// TwinCAT 3 PLC project PRG_B_BaseDecorator
// Title: B_BaseDecorate
// Company: RafalOS
// Author: Rafał Osajda
// ProjectVersion: 0.0.0.3
// ProgramVersion: 3.1.4024.0
// libraries:
//   B_Base, * (RafalOS)
//   Tc2_Standard, * (Beckhoff Automation GmbH)
//   Tc2_System, * (Beckhoff Automation GmbH)
//   Tc3_Module, * (Beckhoff Automation GmbH)
// project tree:
//   / PlcTask.TcTTO
//   POUs Compilation/ PRG_Compilation.TcPOU
//   POUs/A03_FB_BaseLoggerElementDecorator/ FB_BaseLoggerElementDecoratorParent.TcPOU (not stored), ITF_BaseLoggerElementDecoratorParent.TcIO (not stored)
//   POUs/A04_FB_BaseComponentDecorator/ FB_BaseComponentDecoratorParent.TcPOU (not stored), ITF_BaseComponentDecoratorParent.TcIO
//   POUs/A05_FB_BaseControlElementDecorator/ FB_BaseControlElementDecoratorParent.TcPOU (not stored), ITF_BaseControlElementDecoratorParent.TcIO (not stored)
//   POUs/A06_FB_BaseGroupElementDecorator/ FB_BaseGroupElementDecoratorParent.TcPOU (not stored), ITF_BaseGroupElementDecoratorParent.TcIO
//   POUs/A07_FB_BaseTopElementDecorator/ FB_BaseTopElementDecoratorParent.TcPOU (not stored), ITF_BaseTopElementDecoratorParent.TcIO (not stored)

CONFIGURATION PRG_B_BaseDecorator
    RESOURCE PLC ON TwinCAT3
        TASK PlcTask(INTERVAL := T#10ms, PRIORITY := 20);
        PROGRAM PRG_Compilation WITH PlcTask : PRG_Compilation;
    END_RESOURCE
END_CONFIGURATION

// ---- POUs/A04_FB_BaseComponentDecorator/ITF_BaseComponentDecoratorParent.TcIO
INTERFACE ITF_BaseComponentDecoratorParent EXTENDS ITF_BaseComponent

END_INTERFACE

// ---- POUs/A06_FB_BaseGroupElementDecorator/ITF_BaseGroupElementDecoratorParent.TcIO
INTERFACE ITF_BaseGroupElementDecoratorParent EXTENDS ITF_BaseGroupElement

END_INTERFACE

// ---- POUs Compilation/PRG_Compilation.TcPOU
PROGRAM PRG_Compilation
VAR
	fbLoggerElement				: FB_BaseLoggerElement;
	fbLoggerElementDecorator	: FB_BaseLoggerElementDecoratorParent (fbToDecorate := fbLoggerElement);
	fbComponent					: FB_BaseComponent;
	fbComponentDecorator		: FB_BaseComponentDecoratorParent (fbToDecorate := fbComponent);
	fbControlElement			: FB_BaseControlElement;
	fbControlElementDecorator	: FB_BaseControlElementDecoratorParent (fbToDecorate := fbControlElement);
	fbGroupElement				: FB_BaseGroupElement;
	fbGroupElementDecorator		: FB_BaseGroupElementDecoratorParent (fbToDecorate := fbGroupElement);
	fbTopElement				: FB_BaseTopElement;
	fbTopElementDecorate		: FB_BaseTopElementDecoratorParent (fbToDecorate := fbTopElement);
END_VAR

END_PROGRAM
